// TwinCAT 3 PLC project Tc3_XL_Moition
// Title: Tc3_XL_Motion
// Company: Beckhoff Automation GmbH
// Author: H Kühlmann
// ProjectVersion: 0.0.1.26
// Description: Base Functions für XL
// ProgramVersion: 3.1.4026.13
// libraries:
//   Tc2_Standard, * (Beckhoff Automation GmbH)
//   Tc3_EventLogger, * (Beckhoff Automation GmbH)
//   Tc3_Mc3PlanarMotion, * (Beckhoff Automation GmbH)
//   Tc3_Module, * (Beckhoff Automation GmbH)
//   Tc3_Physics, * (Beckhoff Automation GmbH)
//   Tc3_XtsInterface,newest,Beckhoff Automation GmbH
// project tree:
//   Mover/DUTs/ E_TrackNum.TcDUT, ST_MoverInfo.TcDUT, ST_MoverOnTrackInfo.TcDUT, ST_PointerAddresses.TcDUT, ST_ScopeValues.TcDUT
//   Mover/ITFs/ I_Mover.TcIO
//   Mover/POUs/ FB_Mover.TcPOU
//   Version/ Global_Version.TcGVL

// ---- Mover/DUTs/E_TrackNum.TcDUT
{attribute 'qualified_only'}
{attribute 'strict'}
{attribute 'to_string'}
TYPE E_TrackNum :
	(
	MainStart 	:= 1,	
	Big 		:= 2,
	MainEnd		:= 3,
	Small 		:= 4);	
END_TYPE

// ---- Mover/DUTs/ST_MoverInfo.TcDUT
TYPE ST_MoverInfo :
STRUCT

	MoverOtcid :  Otcid;
	IsVirtuell : BOOL;
	IsActive : BOOL;
	ActPos: LREAL;
	ActVelo: LREAL;
	PlanarMoverCommandMode :STRING(30);// MC_Planar_Mover_Command_Mode;
	State : STRING(20);//MC_Planar_State;
	Positition : LREAL;
	Track :STRING(20);
	Error: BOOL;
	ErrorID : UDINT;
	TargetTrackPosition  : LREAL;
	TargetTrack : Otcid;
	RemainingDistance : LREAL;
	Gap : LREAL;
	LimitVelo : LREAL; 
	LimitAcc : LREAL;
	LimitDec : LREAL;
	LimitJerk : LREAL;
	
END_STRUCT
END_TYPE

// ---- Mover/DUTs/ST_MoverOnTrackInfo.TcDUT
TYPE ST_MoverOnTrackInfo :
STRUCT
	TargetPosition 		: LREAL;
	TargetTrack 		: Otcid;
	Remainingdistance 	: LREAL;
	Gap 				: LREAL;
	LimitV 				: LREAL;
	LimitA 				: LREAL;
	LimitD 				: LREAL;
	LimitJ 				: LREAL;
	GapMode				: MC.MC_GAP_MODE_ON_TRACK;
	DynamicMode			: MC.MC_DYNAMIC_MODE_ON_TRACK;
	Movementtype		: MC.MC_MOVEMENT_TYPE_ON_TRACK;
END_STRUCT
END_TYPE

// ---- Mover/DUTs/ST_PointerAddresses.TcDUT
TYPE ST_PointerAddresses :
STRUCT
	SetCurrentPointer 		: POINTER TO LREAL;
	ActHwPosModuloPointer 	: POINTER TO LREAL;
	ActPosErrorPointer 		: POINTER TO LREAL;
	SetVeloItpPointer		: POINTER TO LREAL;
	SetAccItpPointer	 	: POINTER TO LREAL;
	ActVeloPointer 			: POINTER TO LREAL;
	SetForcePointer			: POINTER TO LREAL;

END_STRUCT
END_TYPE

// ---- Mover/DUTs/ST_ScopeValues.TcDUT
TYPE ST_ScopeValues :
STRUCT
	SetCurrent 		: LREAL;
	ActHwPosModulo 	: LREAL;
	ActPosError		: LREAL;
	SetVeloItp		: LREAL;
	SetAccItp	 	: LREAL;
	ActVelo 		: LREAL;
	SetForce		: LREAL;
	ActStatus		: driveState;
END_STRUCT
END_TYPE

// ---- Version/Global_Version.TcGVL
{attribute 'TcGenerated'}
{attribute 'no-analysis'}
{attribute 'linkalways'}
// This function has been automatically generated from the project information.
VAR_GLOBAL CONSTANT
	{attribute 'const_non_replaced'}
	stLibVersion_Tc3_XL_Motion : ST_LibVersion := (iMajor := 0, iMinor := 0, iBuild := 1, iRevision := 26, nFlags := 0, sVersion := '0.0.1.26');
END_VAR

// ---- Mover/ITFs/I_Mover.TcIO

INTERFACE I_Mover

METHOD CycleUpdate : BOOL
VAR_INPUT
END_VAR
END_METHOD

METHOD Disable : bool
VAR_INPUT
END_VAR
END_METHOD

METHOD Enable : bool
VAR_INPUT
END_VAR
END_METHOD

METHOD GetDistanceToEot : LREAL
VAR_INPUT
	TrackLenght : LREAL;
END_VAR
END_METHOD

METHOD Halt : bool
VAR_INPUT
END_VAR
END_METHOD

METHOD Init : BOOL
VAR_INPUT
	XtsMover:  I_XtsXlMover1;
	XtsProcessingUnit :  I_XtsProcessingUnit1;

	
END_VAR
END_METHOD

METHOD JoinNearestTrack : BOOL

VAR_INPUT 
	aMcTracks : ARRAY[*] OF MC_PlanarTrack;
	Trackcount : UINT;
END_VAR
END_METHOD

METHOD LeaveSystemAt : BOOL
VAR_INPUT
	ConnectionOut: REFERENCE TO MC_PlanarTrackConnectionOut;	
	gap : LREAL; 		
END_VAR
END_METHOD

METHOD MoveOnTrack : BOOL
VAR_INPUT
	track: REFERENCE TO MC_PlanarTrack;	
	targetPos: LREAL;
	gap : LREAL; 

END_VAR
END_METHOD

PROPERTY MoverStopped : BOOL
GET
END_GET
SET
END_SET
END_PROPERTY

PROPERTY P_Dynamics : REFERENCE TO DynamicConstraint_PathXY;
GET
END_GET
END_PROPERTY

PROPERTY P_IsInitialized : bool
GET
END_GET
END_PROPERTY

PROPERTY P_MoverOTCID : OTCID
GET
END_GET
SET
END_SET
END_PROPERTY

PROPERTY P_PlanarFeedback : REFERENCE TO MC_PlanarFeedback
GET
END_GET
END_PROPERTY

PROPERTY P_PlanarMover :   REFERENCE TO  MC_PlanarMover
GET
END_GET
END_PROPERTY

PROPERTY P_SyncFeedback :  REFERENCE TO MC_PlanarFeedbackGearInPosOnTrackWithMasterMover
GET
END_GET
END_PROPERTY

PROPERTY P_TargetTrack : UDINT
GET
END_GET
SET
END_SET
END_PROPERTY

PROPERTY Rework : BOOL
GET
END_GET
SET
END_SET
END_PROPERTY

METHOD SyncToOtherMover : Bool
VAR_INPUT
	masterSyncPos : LREAL; // Position on the master track
	followerSyncPos : LREAL; // position on the follower track
	PlanarMoverToFollow: REFERENCE TO Tc3_Mc3PlanarMotion.MC_PlanarMover;
	masterTrack : REFERENCE TO Tc3_Mc3PlanarMotion.MC_PlanarTrack; 
	followerTrack : REFERENCE TO Tc3_Mc3PlanarMotion.MC_PlanarTrack; 
	velo :  REFERENCE TO LREAL; 
END_VAR
END_METHOD

METHOD  UpdateXtsTrack
VAR_INPUT
END_VAR
VAR

END_VAR
END_METHOD

PROPERTY XlProcessingUnit : I_XtsProcessingUnit1
GET
END_GET
END_PROPERTY

PROPERTY XtsComFeed : REFERENCE TO  XtsCommandFeedback
GET
END_GET
END_PROPERTY

PROPERTY XtsXlMover :  I_XtsXlMover1
GET
END_GET
END_PROPERTY

END_INTERFACE

// ---- Mover/POUs/FB_Mover.TcPOU
{attribute 'no_assign'}
FUNCTION_BLOCK FB_Mover IMPLEMENTS I_Mover
VAR_INPUT
END_VAR
VAR_OUTPUT
END_VAR
VAR
	_bIsInitialized: BOOL;	

	fbPlanarMover : MC_PlanarMover;
	fbPlanarFeedback: MC_PlanarFeedback;
	trackTrail: MC_PlanarTrackTrail;
	SyncMoverFeedback: Tc3_Mc3PlanarMotion.MC_PlanarFeedbackGearInPosOnTrackWithMasterMover;
	
	_GearInOptions: Tc3_Mc3PlanarMotion.ST_GearInPosOnTrackWithMasterMoverOptions;
	_stMoveOnTrackOptions: ST_MoveOnTrackOptions;
	_stLeaveSystemAtOptions : ST_LeaveSystemAtOptions;
	
	_syncTrail : MC_PlanarTrackTrail;
	
	CmdFeedback :  XtsCommandFeedback;
	ipXtsMover:   I_XtsXlMover1;
	ipXtsProcessingUnit:  I_XtsProcessingUnit1;

	_stMoverInfos : ST_MoverInfo;	
	_stMoverOnTrackInfos : MC_MOVER_ON_TRACK_INFORMATION;

	_nextMcTrackOid: OTCID;
	_stDynamics: DynamicConstraint_PathXY;
	_TargetTrack : UDINT;
	_ReWork : BOOL;
	_partConfig: UINT;
	_InSync :BOOL; 
	_PositionOnTrack : LREAL;
	_Track : OTCID; 
	_distToEndOfTrack : LREAL;

	fbResult						: FB_TcMessage;
///	_ipComObject					: ITComObject;
	PID_OnTrackInfos				: PTCID := 16#05030180;
	bInit 							: BOOL;
	nErrorID						: HRESULT; 
	ControllerOID					: otcid;
	stPointerAddresses				: ST_PointerAddresses;
	ScopeVariables					: ST_ScopeValues;
	
END_VAR

METHOD ClearSyncTrail : BOOL
VAR_INPUT
END_VAR
_syncTrail.Clear();

IF _syncTrail.TrackCount = 0 THEN
	ClearSyncTrail := TRUE;
END_IF
END_METHOD



METHOD CycleUpdate : BOOL


VAR_INST
	_trackEnum: e_TrackNum;

END_VAR
IF NOT _bIsInitialized THEN
	RETURN;
END_IF

fbPlanarMover.GetTrackTrailInformation(trackTrail);
_PositionOnTrack := fbPlanarMover.MCTOPLC.SETONTRACK.SetPos;


fbPlanarMover.Update();
fbPlanarFeedback.Update();
SyncMoverFeedback.Update();
UpdateXtsTrack();
GetOnTrackInfos(fbPlanarMover.MCTOPLC.STD.MoverOID) ;


_stMoverinfos.MoverOtcid :=fbPlanarMover.MCTOPLC.STD.MoverOID ;
_stMoverinfos.IsActive := ipXtsMover.GetIsActive(0);
_stMoverinfos.ActPos :=  ipXtsMover.GetPositionInfo_trackPosition(0);
_stMoverinfos.ActVelo := fbPlanarMover.MCTOPLC.SETONTRACK.SetVelo;
_stMoverinfos.IsVirtuell := ipXtsMover.GetIsVirtualFeedbackEnabled(0);
_stMoverinfos.Positition :=	fbPlanarMover.MCTOPLC.SETONTRACK.SetPos;
_stMoverinfos.Track := TO_STRING(_trackEnum);
_stMoverinfos.Error := fbPlanarMover.Error;
_stMoverinfos.ErrorID := fbPlanarMover.ErrorId;
_stMoverinfos.PlanarMoverCommandMode :=  TO_STRING(fbPlanarMover.MCTOPLC.STD.CommandMode);
_stMoverinfos.State :=  TO_STRING(fbPlanarMover.MCTOPLC.STD.State);
_stMoverinfos.Gap := _stMoverOnTrackInfos.Gap;
_stMoverinfos.LimitAcc := _stMoverOnTrackInfos.Limits.A;
_stMoverinfos.LimitDec := _stMoverOnTrackInfos.Limits.D;
_stMoverinfos.LimitJerk := _stMoverOnTrackInfos.Limits.J;
_stMoverinfos.LimitVelo := _stMoverOnTrackInfos.Limits.V;
_stMoverinfos.TargetTrackPosition := _stMoverOnTrackInfos.TargetPosition.Position;
_stMoverinfos.TargetTrack := _stMoverOnTrackInfos.TargetPosition.TrackOid;
_stMoverinfos.RemainingDistance := _stMoverOnTrackInfos.Remainingdistance;
ScopeVariables.ActStatus := ipXtsMover.GetDriveStatus(0);
IF stPointerAddresses.ActHwPosModuloPointer <> 0 THEN
	ScopeVariables.ActHwPosModulo := stPointerAddresses.ActHwPosModuloPointer^ ;
	ScopeVariables.ActPosError := stPointerAddresses.ActPosErrorPointer^ ;
	ScopeVariables.ActVelo := stPointerAddresses.ActVeloPointer^ ;
	ScopeVariables.SetAccItp := stPointerAddresses.SetAccItpPointer^;
	ScopeVariables.SetCurrent := stPointerAddresses.SetCurrentPointer^ ;
	ScopeVariables.SetVeloItp := stPointerAddresses.SetVeloItpPointer^  ;
	ScopeVariables.SetForce := stPointerAddresses.SetForcePointer^;

END_IF
END_METHOD

METHOD Disable : BOOL
VAR_INPUT
END_VAR
fbPlanarMover.Enable(
	commandFeedback:= fbPlanarFeedback);
	
Disable :=fbPlanarFeedback.Done OR fbPlanarFeedback.Error;
END_METHOD

METHOD Enable : BOOL
VAR_INPUT
END_VAR
fbPlanarMover.Disable(
	commandFeedback:= fbPlanarFeedback);
	
Enable :=fbPlanarFeedback.Done OR fbPlanarFeedback.Error;
END_METHOD

METHOD GetActHwPosModuloPointer : POINTER TO LREAL
VAR_INPUT
	ControllerOID : OTCID;
END_VAR
VAR
	ipComObject			: ITcWatchSource;
	oidActHwPosModulo	: OTCID := 16#A0000010;
	sizeData			: UDINT;
	adrData 			: PVOID; 
END_VAR

nErrorID := FW_ObjMgr_GetObjectInstance(	oid		:=	ControllerOID, 
											iid		:=	TC_GLOBAL_IID_LIST.IID_ITcWatchSource, 
											pipUnk 	:= ADR(ipComObject));


																				
IF ipComObject <> 0 THEN
	
	sizeData := SIZEOF(GetActHwPosModuloPointer);
	adrData := ADR(GetActHwPosModuloPointer);

	nErrorID := ipComObject.InterpretGroupOffsetLength( 	indexOffset := oidActHwPosModulo ,
															cbLength 	:= sizeData,
															ppData 		:= adrData);
	ipComObject.TcRelease();	
	ipComObject := 0;													
														
												
END_IF
END_METHOD

METHOD GetActPosErrorPointer : POINTER TO LREAL
VAR_INPUT
	ControllerOID : OTCID;
END_VAR
VAR
	ipComObject			: ITcWatchSource;
	oidActPosError		: OTCID := 16#A0000018;
	sizeData			: UDINT;
	adrData 			: PVOID; 
END_VAR

nErrorID := FW_ObjMgr_GetObjectInstance(	oid		:=	ControllerOID, 
											iid		:=	TC_GLOBAL_IID_LIST.IID_ITcWatchSource, 
											pipUnk 	:= ADR(ipComObject));


																				
IF ipComObject <> 0 THEN
	
	sizeData := SIZEOF(GetActPosErrorPointer);
	adrData := ADR(GetActPosErrorPointer);

	nErrorID := ipComObject.InterpretGroupOffsetLength( 	indexOffset := oidActPosError ,
															cbLength 	:= sizeData,
															ppData 		:= adrData);
	ipComObject.TcRelease();	
	ipComObject := 0;													
														
												
END_IF
END_METHOD

METHOD GetActVeloPointer : POINTER TO LREAL
VAR_INPUT
	ControllerOID : OTCID;
END_VAR
VAR
	ipComObject			: ITcWatchSource;
	oidActVelo	: OTCID := 16#A0000008;
	sizeData			: UDINT;
	adrData 			: PVOID; 
END_VAR

nErrorID := FW_ObjMgr_GetObjectInstance(	oid		:=	ControllerOID, 
											iid		:=	TC_GLOBAL_IID_LIST.IID_ITcWatchSource, 
											pipUnk 	:= ADR(ipComObject));


																				
IF ipComObject <> 0 THEN
	
	sizeData := SIZEOF(GetActVeloPointer);
	adrData := ADR(GetActVeloPointer);

	nErrorID := ipComObject.InterpretGroupOffsetLength( 	indexOffset := oidActVelo ,
															cbLength 	:= sizeData,
															ppData 		:= adrData);
	ipComObject.TcRelease();	
	ipComObject := 0;													
														
												
END_IF
END_METHOD

METHOD GetDistanceToEot : LREAL
VAR_INPUT
	TrackLenght : LREAL;
END_VAR
GetDistanceToEot := _distToEndOfTrack;

IF fbPlanarMover.MCTOPLC.SETONTRACK.TrackOID<>0 THEN 
	GetDistanceToEot := TrackLenght-fbPlanarMover.MCTOPLC.SETONTRACK.SetPos;
END_IF
END_METHOD

METHOD GetOnTrackInfos : BOOL
VAR_INPUT
	nObjectId : otcid; 
END_VAR
VAR
	nData 			: UDINT := SIZEOF(_stMoverOnTrackInfos);
	pData 			: PVOID := ADR(_stMoverOnTrackInfos);
	stEventEntry	: TcEventEntry;
	pstEventEntry	: REFERENCE TO TcEventEntry REF= stEventEntry;
END_VAR
VAR_INST
	hResult : HRESULT;
	bError : BOOL;
	_ipComObject : ITComObject;
END_VAR
bError := FALSE;


IF nObjectId <> 0 AND_THEN _ipComObject = 0 THEN
	 FW_ObjMgr_GetObjectInstance(	oid		:= nObjectId, 
								iid		:= TC_GLOBAL_IID_LIST.IID_ITComObject, 
								pipUnk	:= ADR(_ipComObject)) ;
END_IF

IF _ipComObject <> 0 THEN 
	 hResult := 	_ipComObject.TcgetObjPara(		pid := PID_OnTrackInfos,
													nData := nData,
													pData := pData,
													pgp := 0); 	
	IF hResult = 0 THEN
		GetOnTrackInfos := TRUE;
ELSE
	HRESULTAdsErr_TO_TcEventEntry(hResult,stEventEntry);
	IF NOT fbResult.EqualsToEventEntryEx( stOther := stEventEntry) THEN
		fbResult.CreateEx(stEventEntry, 0);
		fbResult.Send(0);
		fbResult.Release();
	END_IF
		bError := TRUE;
	END_IF							
END_IF
END_METHOD

METHOD GetSetAccItpPointer : POINTER TO LREAL
VAR_INPUT
	ControllerOID : OTCID;
END_VAR
VAR
	ipComObject			: ITcWatchSource;
	oidSetAccItp		: OTCID := 16#A0000038;
	sizeData			: UDINT;
	adrData 			: PVOID; 
END_VAR

nErrorID := FW_ObjMgr_GetObjectInstance(	oid		:=	ControllerOID, 
											iid		:=	TC_GLOBAL_IID_LIST.IID_ITcWatchSource, 
											pipUnk 	:= ADR(ipComObject));


																				
IF ipComObject <> 0 THEN
	
	sizeData := SIZEOF(GetSetAccItpPointer);
	adrData := ADR(GetSetAccItpPointer);

	nErrorID := ipComObject.InterpretGroupOffsetLength( 	indexOffset := oidSetAccItp ,
															cbLength 	:= sizeData,
															ppData 		:= adrData);
	ipComObject.TcRelease();	
	ipComObject := 0;													
														
												
END_IF
END_METHOD

METHOD GetSetCurrentPointer : POINTER TO LREAL
VAR_INPUT
	ControllerOID : OTCID;
END_VAR
VAR
	ipComObject			: ITcWatchSource;
	oidSetCurrent 		: OTCID := 16#A0000048;
	sizeData			: UDINT;
	adrData 			: PVOID; 
END_VAR

nErrorID := FW_ObjMgr_GetObjectInstance(	oid		:=	ControllerOID, 
											iid		:=	TC_GLOBAL_IID_LIST.IID_ITcWatchSource, 
											pipUnk 	:= ADR(ipComObject));


																				
IF ipComObject <> 0 THEN
	
	sizeData := SIZEOF(GetSetCurrentPointer);
	adrData := ADR(GetSetCurrentPointer);

	nErrorID := ipComObject.InterpretGroupOffsetLength( 	indexOffset := oidSetCurrent ,
															cbLength 	:= sizeData,
															ppData 		:= adrData);
	ipComObject.TcRelease();	
	ipComObject := 0;													
														
												
END_IF
END_METHOD

METHOD GetSetForcePointer : POINTER TO LREAL
VAR_INPUT
	ControllerOID : OTCID;
END_VAR
VAR
	ipComObject			: ITcWatchSource;
	oidSetForce 		: OTCID := 16#A0000050;
	sizeData			: UDINT;
	adrData 			: PVOID; 
END_VAR

nErrorID := FW_ObjMgr_GetObjectInstance(	oid		:=	ControllerOID, 
											iid		:=	TC_GLOBAL_IID_LIST.IID_ITcWatchSource, 
											pipUnk 	:= ADR(ipComObject));


																				
IF ipComObject <> 0 THEN
	
	sizeData := SIZEOF(GetSetForcePointer);
	adrData := ADR(GetSetForcePointer);

	nErrorID := ipComObject.InterpretGroupOffsetLength( 	indexOffset := oidSetForce ,
															cbLength 	:= sizeData,
															ppData 		:= adrData);
	ipComObject.TcRelease();	
	ipComObject := 0;													
														
												
END_IF
END_METHOD

METHOD GetSetVeloItpPointer : POINTER TO LREAL
VAR_INPUT
	ControllerOID : OTCID;
END_VAR
VAR
	ipComObject			: ITcWatchSource;
	oidSetVeloItp	: OTCID := 16#A0000030;
	sizeData			: UDINT;
	adrData 			: PVOID; 
END_VAR

nErrorID := FW_ObjMgr_GetObjectInstance(	oid		:=	ControllerOID, 
											iid		:=	TC_GLOBAL_IID_LIST.IID_ITcWatchSource, 
											pipUnk 	:= ADR(ipComObject));


																				
IF ipComObject <> 0 THEN
	
	sizeData := SIZEOF(GetSetVeloItpPointer);
	adrData := ADR(GetSetVeloItpPointer);

	nErrorID := ipComObject.InterpretGroupOffsetLength( 	indexOffset := oidSetVeloItp ,
															cbLength 	:= sizeData,
															ppData 		:= adrData);
	ipComObject.TcRelease();	
	ipComObject := 0;													
														
												
END_IF
END_METHOD

METHOD Halt : BOOL
VAR_INPUT
END_VAR
fbPlanarMover.Halt(
	commandFeedback:= fbPlanarFeedback, 
	constraint:= _stDynamics);
	
Halt :=fbPlanarFeedback.Done OR fbPlanarFeedback.Error;
END_METHOD

METHOD Init : BOOL
VAR_INPUT

	XtsMover:   I_XtsXlMover1;
	XtsProcessingUnit :  I_XtsProcessingUnit1;

	
END_VAR
VAR_STAT
	Getpointer : BOOL;
END_VAR


ipXtsMover:= XtsMover;
ipXtsProcessingUnit :=  XtsProcessingUnit;




ControllerOID:= ipXtsMover.GetMoverController(CmdFeedback);
IF ControllerOID <> 0  THEN
	stPointerAddresses.ActHwPosModuloPointer := GetActHwPosModuloPointer(ControllerOID);
	stPointerAddresses.SetVeloItpPointer := GetSetVeloItpPointer(ControllerOID);
	stPointerAddresses.ActVeloPointer := GetActVeloPointer(ControllerOID);
	stPointerAddresses.SetAccItpPointer := GetSetAccItpPointer(ControllerOID);
	stPointerAddresses.ActPosErrorPointer := GetActPosErrorPointer(ControllerOID);
	stPointerAddresses.SetCurrentPointer := GetSetCurrentPointer(ControllerOID); 
	stPointerAddresses.SetForcePointer := GetSetForcePointer(ControllerOID); 
	bInit:=TRUE;
	
	
END_IF
			
IF    CmdFeedback.IsDone THEN
	_bIsInitialized := TRUE;
	Init := TRUE;
END_IF
END_METHOD

METHOD JoinNearestTrack : BOOL
VAR_INPUT 
	aMcTracks : ARRAY[*] OF MC_PlanarTrack;
	Trackcount : UINT;
END_VAR

VAR_INST
	nForCounter: UINT;
	mcTrackOid: OTCID;
	partOid: OTCID;
	cmdFeedback					: 	XtsCommandFeedback;
	objectInfo: PlanarObjectInfo;
END_VAR
partOid := ipXtsMover.GetPositionInfo_partObjectId(cmdFeedback);

IF partOid = 0 THEN
	RETURN;
END_IF

IF cmdFeedback.IsDone THEN
	mcTrackOid := ipXtsProcessingUnit.XlPartWithOid(partOid, cmdFeedback).GetMcTrackOid(cmdFeedback);
	
	FOR nForCounter := 1 TO Trackcount DO
		objectInfo := aMcTracks[nForCounter].GetPlanarObjectInfo();
		IF objectInfo.Id = mcTrackOid THEN
			fbPlanarMover.JoinTrack(fbPlanarFeedback, aMcTracks[nForCounter], _stDynamics, 0); 
			RETURN;
		END_IF
	END_FOR
END_IF
END_METHOD

METHOD LeaveSystemAt : BOOL
VAR_INPUT
	ConnectionOut: REFERENCE TO MC_PlanarTrackConnectionOut;
	gap : LREAL; 
END_VAR
_stLeaveSystemAtOptions.gap := gap;
_stLeaveSystemAtOptions.gapMode := MC_GAP_MODE_ON_TRACK.Fast1D; 
_stLeaveSystemAtOptions.dynamicMode :=  MC_DYNAMIC_MODE_ON_TRACK.None;

fbPlanarMover.LeaveSystemAt(fbPlanarFeedback, ConnectionOut,  _stDynamics,_stLeaveSystemAtOptions);
END_METHOD

METHOD MoveOnTrack : BOOL
VAR_INPUT
	track: REFERENCE TO MC_PlanarTrack;	
	targetPos: LREAL;
	gap : LREAL; 
END_VAR
_stMoveonTrackOptions.gap := gap; 

fbPlanarMover.MoveOnTrack(
	commandFeedback:= fbPlanarFeedback, 
	targetTrack:= track, 
	targetPositionOnTrack:= targetPos, 
	constraint:= _stDynamics, 
	options:= _stMoveOnTrackOptions);
END_METHOD

PROPERTY MoverStopped : BOOL
GET
MoverStopped := (fbPlanarMover.MCTOPLC.SETONTRACK.SetVelo < 20);
END_GET
SET
END_SET
END_PROPERTY

PROPERTY P_Dynamics : REFERENCE TO DynamicConstraint_PathXY;
GET

P_Dynamics REF= _stDynamics;
END_GET
END_PROPERTY

PROPERTY P_IsInitialized : bool
GET
P_IsInitialized := _bIsInitialized;
END_GET
END_PROPERTY

PROPERTY P_MoveOnTrackOptions  : REFERENCE TO  ST_MoveOnTrackOptions
GET
P_MoveOnTrackOptions REF= _stMoveOnTrackOptions;
END_GET
END_PROPERTY

PROPERTY P_MoverInfos : REFERENCE TO ST_MoverInfo
GET
P_MoverInfos  REF= _stMoverInfos;
END_GET
END_PROPERTY

PROPERTY p_MoverOTCID : OTCID
GET
p_MoverOTCID := fbPlanarMover.MCTOPLC.STD.MoverOID;
END_GET
SET
END_SET
END_PROPERTY

PROPERTY P_PlanarFeedback : REFERENCE TO MC_PlanarFeedback
GET
P_PlanarFeedback REF= fbPlanarFeedback;
END_GET
END_PROPERTY

PROPERTY P_PlanarMover :   REFERENCE TO  MC_PlanarMover
GET
P_PlanarMover REF= fbPlanarMover;
END_GET
END_PROPERTY

PROPERTY P_ScopeVariables  :   REFERENCE TO ST_ScopeValues
GET
 P_ScopeVariables   REF= ScopeVariables;
END_GET
END_PROPERTY

PROPERTY P_SyncFeedback :  REFERENCE TO MC_PlanarFeedbackGearInPosOnTrackWithMasterMover
GET
P_SyncFeedback REF= SyncMoverFeedback;
END_GET
END_PROPERTY

PROPERTY P_TargetTrack : UDINT
GET
P_TargetTrack := _TargetTrack ;
END_GET
SET
_TargetTrack := P_TargetTrack;
END_SET
END_PROPERTY

PROPERTY Rework : BOOL
GET
Rework := _Rework;
END_GET
SET
_Rework := Rework;
END_SET
END_PROPERTY

METHOD SetSyncTrail : BOOL
VAR_INPUT
	PlanarTrack : MC_PlanarTrack;
END_VAR
_syncTrail.AddTrack(track:= PlanarTrack);///GVL_Mc.aMCTracks[E_TrackNum.Small]); 
 
SetSyncTrail := TRUE;
END_METHOD

METHOD SyncToOtherMover : BOOL
VAR_INPUT
	masterSyncPos : LREAL; // Position on the master track
	followerSyncPos : LREAL; // position on the follower track
	PlanarMoverToFollow: REFERENCE TO Tc3_Mc3PlanarMotion.MC_PlanarMover;
	masterTrack : REFERENCE TO Tc3_Mc3PlanarMotion.MC_PlanarTrack; 
	followerTrack : REFERENCE TO Tc3_Mc3PlanarMotion.MC_PlanarTrack; 
	velo : REFERENCE TO LREAL; 
END_VAR

VAR
	trail: Tc3_Mc3PlanarMotion.MC_PlanarTrackTrail;

END_VAR
_GearInOptions.allowedSlaveSyncDirections := MC_SYNC_DIRECTIONS.Positive; 
_GearInOptions.directionMasterSyncPosition := MC_DIRECTION.mcDirectionNonModulo; 
_GearInOptions.directionSlaveSyncPosition := MC_DIRECTION.mcDirectionNonModulo;  
_GearInOptions.followMover := FALSE; 
_GearInOptions.gap := 0; // elimnate gap funciton 
_GearInOptions.inSyncToleranceDistance :=0; 
_GearInOptions.moduloToleranceMasterSyncPosition := 0; 
_GearInOptions.moduloToleranceSlaveSyncPosition := 0;  
_stDynamics.V := velo; 

fbPlanarMover.GearInPosOnTrackWithMasterMover(
	commandFeedback:=  SyncMoverFeedback , 
	masterMover:= PlanarMoverToFollow , 
	trackTrail:= _syncTrail, // may need to give a trail maybe not
	masterSyncPosition:= masterSyncPos, 
	masterSyncPositionTrack:= MasterTrack , 
	slaveSyncPosition:= followerSyncPos, 
	slaveSyncPositionTrack:= followerTrack, 
	constraint:=_stDynamics , 
	options:=_GearInOptions );
END_METHOD

METHOD PUBLIC UpdateXtsTrack
VAR_INPUT
END_VAR
VAR_STAT
	nTrackCount: UINT;
	oid1: OTCID;
	oid2: OTCID;
	
	nForCounter: UINT;
	nPartConfigCount: UINT;
	
	partConfig1: OTCID;
	partConfig2: OTCID;
	
	mcTrackOid1: OTCID;
	mcTrackOid2: OTCID;
	trackOid: OTCID;
	
	nTrackTrailCount: UDINT;
	actTrackOid: OTCID;
	nIndexInTrail: UDINT;
END_VAR
nTrackTrailCount := trackTrail.TrackCount;
actTrackOid := fbPlanarMover.MCTOPLC.SETONTRACK.TrackOID;

IF nTrackTrailCount <= 1 THEN
	RETURN;
END_IF

FOR nForCounter := 1 TO UDINT_TO_UINT(nTrackTrailCount) DO
	oid1 := trackTrail.GetTrackOidAt(nForCounter);
	IF oid1 = actTrackOid THEN
		IF nForCounter < nTrackTrailCount THEN
			oid2 := trackTrail.GetTrackOidAt(nForCounter + 1);
			EXIT;
		ELSE
			RETURN; //last one ine track trail
		END_IF
	END_IF
END_FOR

IF oid2 = _nextMcTrackOid AND ipXtsMover.GetPositionInfo_partPosition(CmdFeedback) < 600 THEN //no change
	RETURN;
END_IF

nTrackCount := ipXtsProcessingUnit.TrackCount();

FOR nForCounter := 1 TO nTrackCount DO
	nPartConfigCount := ipXtsProcessingUnit.Track(nForCounter, CmdFeedback).PartConfigCount(); 
	
	IF nPartConfigCount >= 2  THEN
		partConfig1 := ipXtsProcessingUnit.Track(nForCounter, CmdFeedback).GetPartConfigOidAt(1, 0);
		partConfig2 := ipXtsProcessingUnit.Track(nForCounter, CmdFeedback).GetPartConfigOidAt(2, 0);
//
		
		IF partConfig1 = 0 OR partConfig2 = 0 THEN
			CONTINUE;
		END_IF
		
		mcTrackOid1 := ipXtsProcessingUnit.XlPartWithOid(partConfig1, CmdFeedback).GetMcTrackOid(0);
		mcTrackOid2 := ipXtsProcessingUnit.XlPartWithOid(partConfig2, CmdFeedback).GetMcTrackOid(0);
		IF mcTrackOid1 = oid1 AND mcTrackOid2 = oid2   THEN
			trackOid := ipXtsProcessingUnit.Track(nForCounter, CmdFeedback).GetObjectId();
			ipXtsMover.SetActiveTrackObjectId(trackOid, CmdFeedback);
			
			IF CmdFeedback.IsDone THEN
				_nextMcTrackOid := oid2;
			END_IF
			
			RETURN;
		END_IF
	END_IF
END_FOR
END_METHOD

PROPERTY XlProcessingUnit : I_XtsProcessingUnit1
GET
XlProcessingUnit := ipXtsProcessingUnit;
END_GET
END_PROPERTY

PROPERTY XtsComFeed : REFERENCE TO  XtsCommandFeedback
GET
XtsComFeed REF= CmdFeedback;
END_GET
END_PROPERTY

PROPERTY XtsXlMover : I_XtsXlMover1
GET
XtsXlMover := ipXtsMover;
END_GET
END_PROPERTY

END_FUNCTION_BLOCK
